FUNCTION_BLOCK FB_ShortTEST3
VAR_INPUT
	execute: BOOL;
END_VAR
VAR
	TIMERDONE: BOOL;
END_VAR

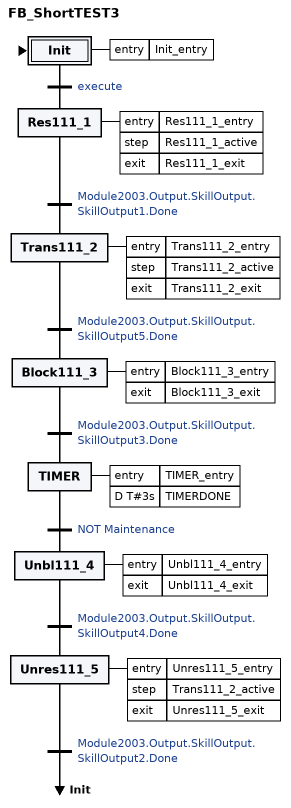
INITIAL_STEP Init:
    Init_entry(P1);  // entry action
END_STEP
TRANSITION FROM Init TO Res111_1
    := execute;
END_TRANSITION
STEP Res111_1:
    Res111_1_entry(P1);  // entry action
    Res111_1_active(N);  // step action
    Res111_1_exit(P0);  // exit action
END_STEP
TRANSITION FROM Res111_1 TO Trans111_2
    := Module2003.Output.SkillOutput.SkillOutput1.Done;
END_TRANSITION
STEP Trans111_2:
    Trans111_2_entry(P1);  // entry action
    Trans111_2_active(N);  // step action
    Trans111_2_exit(P0);  // exit action
END_STEP
TRANSITION FROM Trans111_2 TO Block111_3
    := Module2003.Output.SkillOutput.SkillOutput5.Done;
END_TRANSITION
STEP Block111_3:
    Block111_3_entry(P1);  // entry action
    Block111_3_exit(P0);  // exit action
END_STEP
TRANSITION FROM Block111_3 TO TIMER
    := Module2003.Output.SkillOutput.SkillOutput3.Done;
END_TRANSITION
STEP TIMER:
    TIMER_entry(P1);  // entry action
    TIMERDONE(D, T#3s);
END_STEP
TRANSITION FROM TIMER TO Unbl111_4
    := NOT Maintenance;
END_TRANSITION
STEP Unbl111_4:
    Unbl111_4_entry(P1);  // entry action
    Unbl111_4_exit(P0);  // exit action
END_STEP
TRANSITION FROM Unbl111_4 TO Unres111_5
    := Module2003.Output.SkillOutput.SkillOutput4.Done;
END_TRANSITION
STEP Unres111_5:
    Unres111_5_entry(P1);  // entry action
    Trans111_2_active(N);  // step action
    Unres111_5_exit(P0);  // exit action
END_STEP
TRANSITION FROM Unres111_5 TO Init
    := Module2003.Output.SkillOutput.SkillOutput2.Done;
END_TRANSITION

ACTION Unres111_5_exit:
//unreserve
Module2003.Input.SkillInput.SkillInput2.Execute := FALSE;
Module2003.Input.SkillInput.SkillInput2.ParameterInput.Parameterinput1.Value := 0; //TaskID
END_ACTION

ACTION Block111_3_entry:
//BLOCKIEREN

Module2003.Input.SkillInput.SkillInput3.Execute := TRUE;
Module2003.Input.SkillInput.SkillInput3.ParameterInput.Parameterinput1.Value := 113; //TaskID
END_ACTION

ACTION Res111_1_active:

END_ACTION

ACTION Trans111_2_active:

END_ACTION

ACTION Trans111_2_entry:
//TRANSPORTIEREN

Module2003.Input.SkillInput.SkillInput5.Execute := TRUE;
Module2003.Input.SkillInput.SkillInput5.ParameterInput.Parameterinput1.Value := 169.4; //X-Position
Module2003.Input.SkillInput.SkillInput5.ParameterInput.Parameterinput2.Value := 90; //Z-Position
Module2003.Input.SkillInput.SkillInput5.ParameterInput.Parameterinput3.Value := 400; //Velocity
Module2003.Input.SkillInput.SkillInput5.ParameterInput.Parameterinput4.Value := 100; //Acceleration
END_ACTION

ACTION Unres111_5_entry:
//unreserve
Module2003.Input.SkillInput.SkillInput2.Execute := TRUE;
Module2003.Input.SkillInput.SkillInput2.ParameterInput.Parameterinput1.Value := 113; //TaskID
END_ACTION

ACTION Trans111_6_entry:
//TRANSPORTIEREN

Module2003.Input.SkillInput.SkillInput5.Execute := TRUE;
Module2003.Input.SkillInput.SkillInput5.ParameterInput.Parameterinput1.Value := 20; //X-Position
Module2003.Input.SkillInput.SkillInput5.ParameterInput.Parameterinput2.Value := 80; //Z-Position
Module2003.Input.SkillInput.SkillInput5.ParameterInput.Parameterinput3.Value := 0; //Velocity
Module2003.Input.SkillInput.SkillInput5.ParameterInput.Parameterinput4.Value := 0; //Acceleration
END_ACTION

ACTION Trans111_2_exit:
//TRANSPORTIEREN

Module2003.Input.SkillInput.SkillInput5.Execute := FALSE;
Module2003.Input.SkillInput.SkillInput5.ParameterInput.Parameterinput1.Value := 0; //X-Position
Module2003.Input.SkillInput.SkillInput5.ParameterInput.Parameterinput2.Value := 0; //Z-Position
Module2003.Input.SkillInput.SkillInput5.ParameterInput.Parameterinput3.Value := 0; //Velocity
Module2003.Input.SkillInput.SkillInput5.ParameterInput.Parameterinput4.Value := 0; //Acceleration
END_ACTION

ACTION Init_entry:
execute := FALSE;
END_ACTION

ACTION Res111_1_exit:
// Reservieren entry
Module2003.Input.SkillInput.SkillInput1.Execute := FALSE;
Module2003.Input.SkillInput.SkillInput1.ParameterInput.Parameterinput1.Value := 0; //TASKID
END_ACTION

ACTION TIMER_entry:
TIMERDONE := FALSE;
END_ACTION

ACTION Unbl111_4_entry:
//unBLOCKIEREN

Module2003.Input.SkillInput.SkillInput4.Execute := TRUE; //FALSE weil timer
Module2003.Input.SkillInput.SkillInput4.ParameterInput.Parameterinput1.Value := 112; //TaskID
END_ACTION

ACTION Unbl111_4_exit:
//unBLOCKIEREN

Module2003.Input.SkillInput.SkillInput4.Execute := FALSE; 
Module2003.Input.SkillInput.SkillInput4.ParameterInput.Parameterinput1.Value := 000; //TaskID
END_ACTION

ACTION Trans111_6_exit:
//TRANSPORTIEREN

Module2003.Input.SkillInput.SkillInput5.Execute := FALSE;
Module2003.Input.SkillInput.SkillInput5.ParameterInput.Parameterinput1.Value := 0; //X-Position
Module2003.Input.SkillInput.SkillInput5.ParameterInput.Parameterinput2.Value := 0; //Z-Position
Module2003.Input.SkillInput.SkillInput5.ParameterInput.Parameterinput3.Value := 0; //Velocity
Module2003.Input.SkillInput.SkillInput5.ParameterInput.Parameterinput4.Value := 0; //Acceleration
END_ACTION

ACTION Res111_1_entry:
// Reservieren entry
Module2003.Input.SkillInput.SkillInput1.Execute := TRUE;
Module2003.Input.SkillInput.SkillInput1.ParameterInput.Parameterinput1.Value := 113; //TASKID
END_ACTION

ACTION Block111_3_exit:
//BLOCKIEREN

Module2003.Input.SkillInput.SkillInput3.Execute := FALSE;
Module2003.Input.SkillInput.SkillInput3.ParameterInput.Parameterinput1.Value := 0; //TaskID
END_ACTION

END_FUNCTION_BLOCK

(* stored: Version 1.1.0.1, ProductVersion 3.1.0.25
   POU FB_ShortTEST3: Id {c23f92de-bf05-474f-9d14-4a7cfba99fe4}
   Action Unres111_5_exit: Id {1a603e95-ec44-44e0-942b-b074c05504d6}
   Action Block111_3_entry: Id {1cc36699-11df-4ce0-9b31-0a251cdca354}
   Action Res111_1_active: Id {3e1b94f7-fe74-4b26-a03d-1f647e433245}
   Action Trans111_2_active: Id {47a0d1a0-d78d-4422-ba0b-ac0cb3e4d26b}
   Action Trans111_2_entry: Id {489e286d-43d2-4e77-bb16-c401d0a4c11a}
   Action Unres111_5_entry: Id {4ada7f41-1f7d-4616-b381-96845dd99acb}
   Action Trans111_6_entry: Id {55a69ded-ab81-464d-bd7f-bf24103d63a2}
   Action Trans111_2_exit: Id {565a69b8-d105-4205-949e-cbcc32e28a81}
   Action Init_entry: Id {796a01a1-0f39-463d-9369-efc501ae1dd2}
   Action Res111_1_exit: Id {8fc09498-c219-41f3-af37-6aedf861e73e}
   Action TIMER_entry: Id {a7bf2ba4-08c1-48ae-8e2e-d01e5521c85f}
   Action Unbl111_4_entry: Id {aabb52b6-4abd-45b8-a854-b221c339083f}
   Action Unbl111_4_exit: Id {ad223993-c0bf-426a-87d8-fda7ac41054b}
   Action Trans111_6_exit: Id {c1d61a45-7bfe-4190-a78e-1c4a1ff42560}
   Action Res111_1_entry: Id {c46d397f-a93f-42ca-a78b-fa6a0fdbf28d}
   Action Block111_3_exit: Id {cf4d2419-ff9d-4f76-afdd-3c394cbf5439} *)
